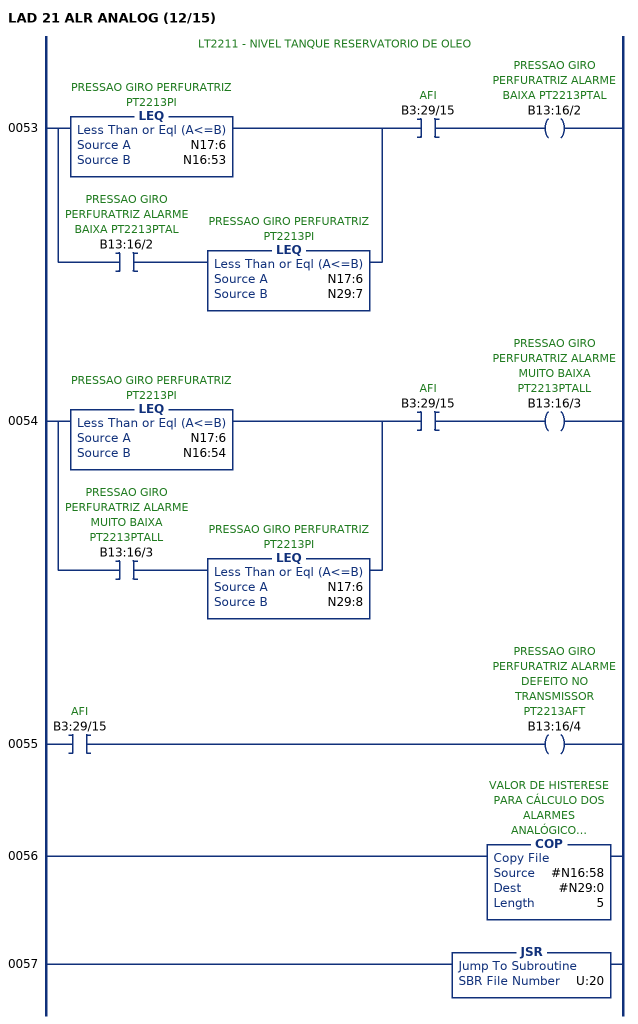
% Rung: 53 %
% LT2211 - NIVEL TANQUE RESERVATORIO DE OLEO %
SOR BST LEQ N17:6 N16:53 NXB XIC B13:16/2 LEQ N17:6 N29:7 BND XIC B3:29/15 OTE B13:16/2 EOR
%   N17:6  PT2213PI  "PRESSAO GIRO PERFURATRIZ" %
%   N16:53  PT2213L  "PRESSAO GIRO PERFURATRIZ BAIXA" %
%   B13:16/2  PT2213PTAL  "PRESSAO GIRO PERFURATRIZ ALARME BAIXA" %
%   N29:7  LIM_AL_L  "LIMITE PARA PERMITIR O REARME DO ALARME L (BAIXO)" %
%   B3:29/15  AFI %
% Rung: 54 %
SOR BST LEQ N17:6 N16:54 NXB XIC B13:16/3 LEQ N17:6 N29:8 BND XIC B3:29/15 OTE B13:16/3 EOR
%   N17:6  PT2213PI  "PRESSAO GIRO PERFURATRIZ" %
%   N16:54  PT2213LL  "PRESSAO GIRO PERFURATRIZ MUITO BAIXA" %
%   B13:16/3  PT2213PTALL  "PRESSAO GIRO PERFURATRIZ ALARME MUITO BAIXA" %
%   N29:8  LIM_AL_LL  "LIMITE PARA PERMITIR O REARME DO ALARME LL (MUITO BAIXO)" %
%   B3:29/15  AFI %
% Rung: 55 %
SOR XIC B3:29/15 OTE B13:16/4 EOR
%   B3:29/15  AFI %
%   B13:16/4  PT2213AFT  "PRESSAO GIRO PERFURATRIZ ALARME DEFEITO NO TRANSMISSOR" %
% Rung: 56 %
SOR COP #N16:58 #N29:0 5 EOR
%   N16:58  LT2211HIS  "NIVEL TANQUE OLEO HISTERESE" %
%   N29:0  HISTERESE  "VALOR DE HISTERESE PARA CÁLCULO DOS ALARMES ANALÓGICOS" %
% Rung: 57 %
SOR JSR U:20 EOR

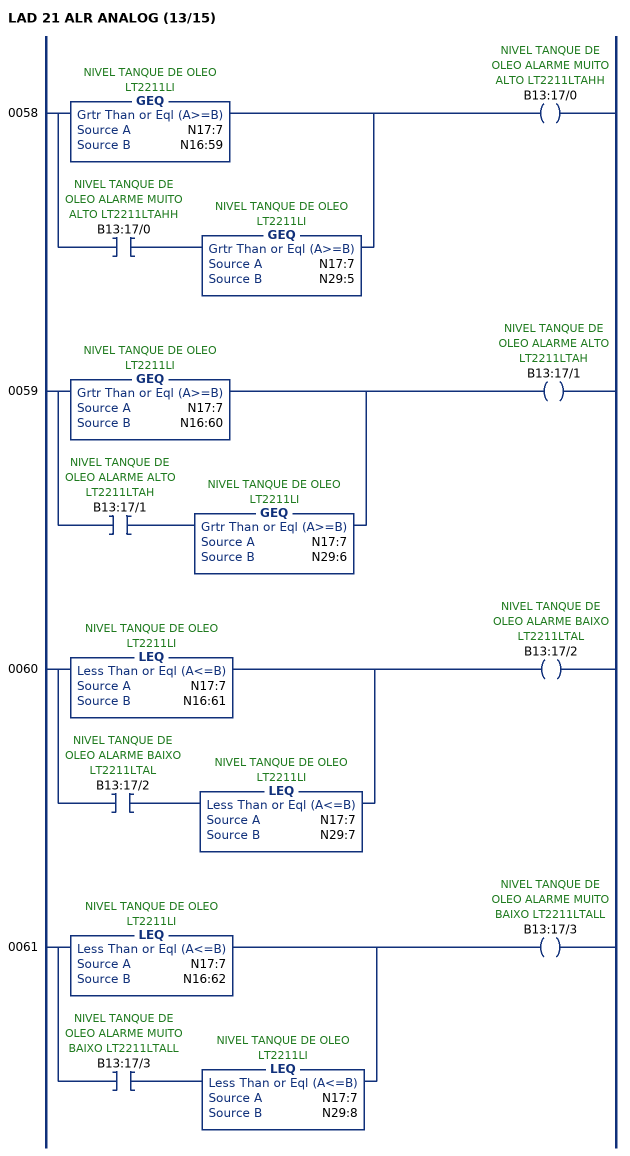
% Rung: 58 %
SOR BST GEQ N17:7 N16:59 NXB XIC B13:17/0 GEQ N17:7 N29:5 BND OTE B13:17/0 EOR
%   N17:7  LT2211LI  "NIVEL TANQUE DE OLEO" %
%   N16:59  LT2211HH  "NIVEL TANQUE OLEO MUITO ALTO" %
%   B13:17/0  LT2211LTAHH  "NIVEL TANQUE DE OLEO ALARME MUITO ALTO" %
%   N29:5  LIM_AL_HH  "LIMITE PARA PERMITIR O REARME DO ALARME HH (MUITO ALTO)" %
% Rung: 59 %
SOR BST GEQ N17:7 N16:60 NXB XIC B13:17/1 GEQ N17:7 N29:6 BND OTE B13:17/1 EOR
%   N17:7  LT2211LI  "NIVEL TANQUE DE OLEO" %
%   N16:60  LT2211H  "NIVEL TANQUE OLEO ALTO" %
%   B13:17/1  LT2211LTAH  "NIVEL TANQUE DE OLEO ALARME ALTO" %
%   N29:6  LIM_AL_H  "LIMITE PARA PERMITIR O REARME DO ALARME H (ALTO)" %
% Rung: 60 %
SOR BST LEQ N17:7 N16:61 NXB XIC B13:17/2 LEQ N17:7 N29:7 BND OTE B13:17/2 EOR
%   N17:7  LT2211LI  "NIVEL TANQUE DE OLEO" %
%   N16:61  LT2211L  "NIVEL TANQUE OLEO BAIXO" %
%   B13:17/2  LT2211LTAL  "NIVEL TANQUE DE OLEO ALARME BAIXO" %
%   N29:7  LIM_AL_L  "LIMITE PARA PERMITIR O REARME DO ALARME L (BAIXO)" %
% Rung: 61 %
SOR BST LEQ N17:7 N16:62 NXB XIC B13:17/3 LEQ N17:7 N29:8 BND OTE B13:17/3 EOR
%   N17:7  LT2211LI  "NIVEL TANQUE DE OLEO" %
%   N16:62  LT2211LL  "NIVEL TANQUE OLEO MUITO BAIXO" %
%   B13:17/3  LT2211LTALL  "NIVEL TANQUE DE OLEO ALARME MUITO BAIXO" %
%   N29:8  LIM_AL_LL  "LIMITE PARA PERMITIR O REARME DO ALARME LL (MUITO BAIXO)" %

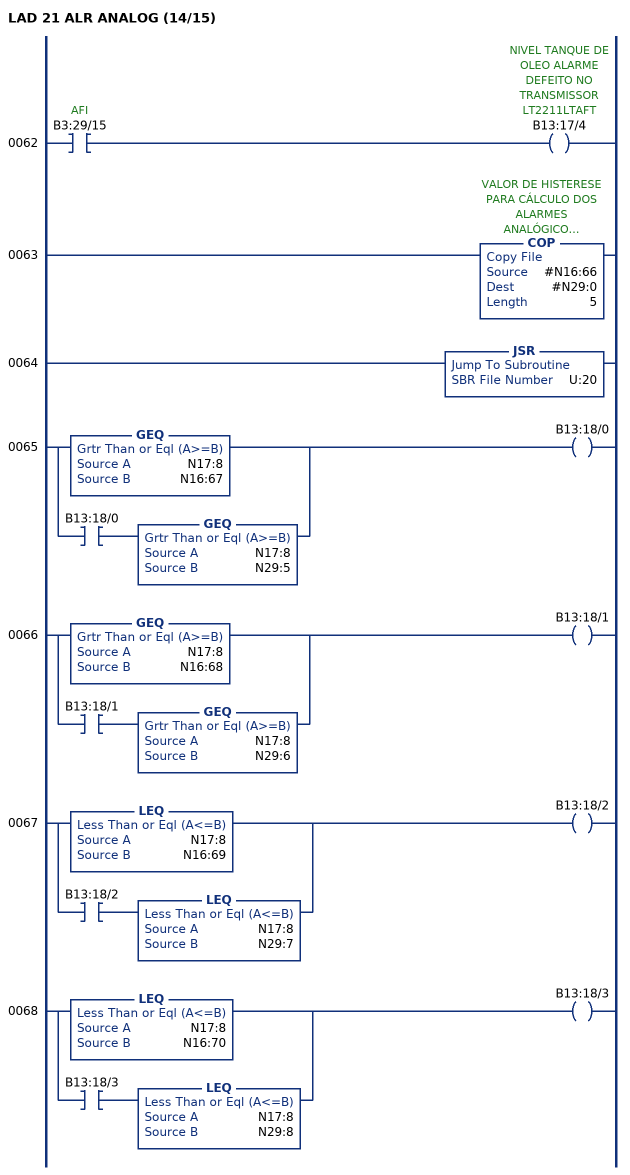
% Rung: 62 %
SOR XIC B3:29/15 OTE B13:17/4 EOR
%   B3:29/15  AFI %
%   B13:17/4  LT2211LTAFT  "NIVEL TANQUE DE OLEO ALARME DEFEITO NO TRANSMISSOR" %
% Rung: 63 %
SOR COP #N16:66 #N29:0 5 EOR
%   N29:0  HISTERESE  "VALOR DE HISTERESE PARA CÁLCULO DOS ALARMES ANALÓGICOS" %
% Rung: 64 %
SOR JSR U:20 EOR
% Rung: 65 %
SOR BST GEQ N17:8 N16:67 NXB XIC B13:18/0 GEQ N17:8 N29:5 BND OTE B13:18/0 EOR
%   N29:5  LIM_AL_HH  "LIMITE PARA PERMITIR O REARME DO ALARME HH (MUITO ALTO)" %
% Rung: 66 %
SOR BST GEQ N17:8 N16:68 NXB XIC B13:18/1 GEQ N17:8 N29:6 BND OTE B13:18/1 EOR
%   N29:6  LIM_AL_H  "LIMITE PARA PERMITIR O REARME DO ALARME H (ALTO)" %
% Rung: 67 %
SOR BST LEQ N17:8 N16:69 NXB XIC B13:18/2 LEQ N17:8 N29:7 BND OTE B13:18/2 EOR
%   N29:7  LIM_AL_L  "LIMITE PARA PERMITIR O REARME DO ALARME L (BAIXO)" %
% Rung: 68 %
SOR BST LEQ N17:8 N16:70 NXB XIC B13:18/3 LEQ N17:8 N29:8 BND OTE B13:18/3 EOR
%   N29:8  LIM_AL_LL  "LIMITE PARA PERMITIR O REARME DO ALARME LL (MUITO BAIXO)" %

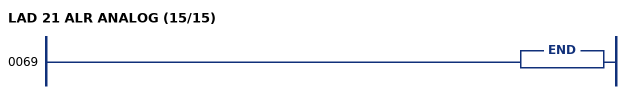
% Rung: 69 %
SOR END EOR

LADDER 22 "UNID ENG"
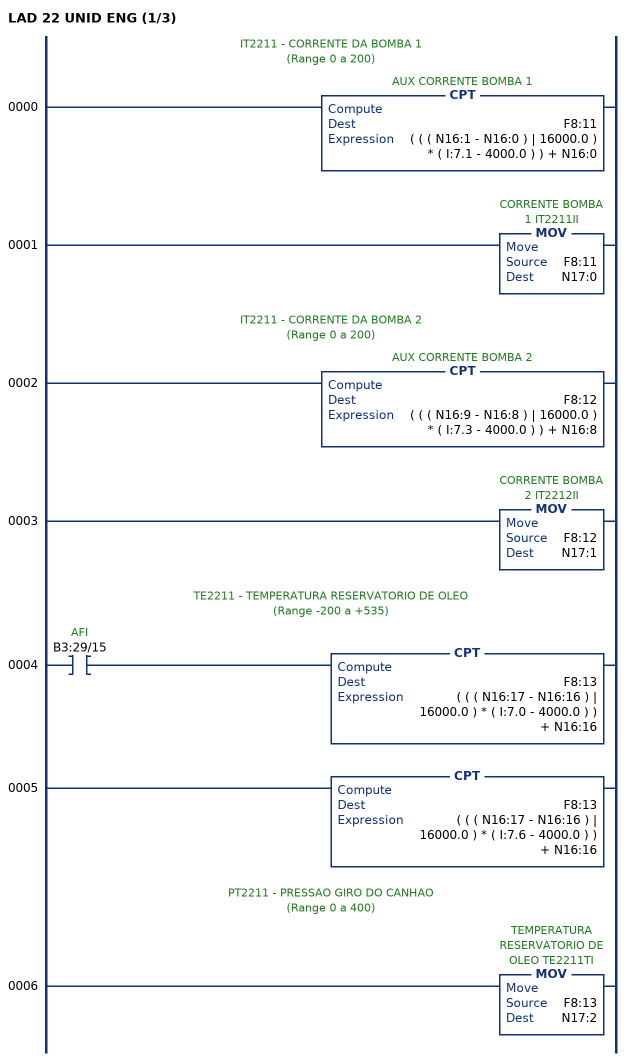
% Rung: 0 %
% IT2211 - CORRENTE DA BOMBA 1
% (Range 0 a 200) %
SOR CPT F8:11 " ( ( ( N16:1 - N16:0 ) | 16000.0 ) * ( I:7.1 - 4000.0 ) ) + N16:0 " EOR
%   F8:11  "AUX CORRENTE BOMBA 1" %
%   N16:1  IT2211MAX  "CORRENTE BOMBA 1 MAXIMO" %
%   N16:0  IT2211MIN  "CORRENTE BOMBA 1 MINIMO" %
%   I:7.1  MT2211  "MOTOR BOMBA 1 MEDICAO DE CORRENTE" %
% Rung: 1 %
SOR MOV F8:11 N17:0 EOR
%   F8:11  "AUX CORRENTE BOMBA 1" %
%   N17:0  IT2211II  "CORRENTE BOMBA 1" %
% Rung: 2 %
% IT2211 - CORRENTE DA BOMBA 2
% (Range 0 a 200) %
SOR CPT F8:12 " ( ( ( N16:9 - N16:8 ) | 16000.0 ) * ( I:7.3 - 4000.0 ) ) + N16:8 " EOR
%   F8:12  "AUX CORRENTE BOMBA 2" %
%   N16:9  IT2212MAX  "CORRENTE BOMBA 2 MAXIMO" %
%   N16:8  IT2212MIN  "CORRENTE BOMBA 2 MINIMO" %
%   I:7.3  MT2213  "MOTOR BOMBA 2 MEDICAO DE CORRENTE" %
% Rung: 3 %
SOR MOV F8:12 N17:1 EOR
%   F8:12  "AUX CORRENTE BOMBA 2" %
%   N17:1  IT2212II  "CORRENTE BOMBA 2" %
% Rung: 4 %
% TE2211 - TEMPERATURA RESERVATORIO DE OLEO
% (Range -200 a +535) %
SOR XIC B3:29/15 CPT F8:13 " ( ( ( N16:17 - N16:16 ) | 16000.0 ) * ( I:7.0 - 4000.0 ) ) + N16:16 " EOR
%   B3:29/15  AFI %
%   N16:17  TE2211MAX  "TEMPERATURA RESERVATORIO DE OLEO MAXIMO" %
%   N16:16  TE2211MIN  "TEMPERATURA RESERVATORIO DE OLEO MINIMO" %
%   I:7.0  TE2211  "TEMPERATURA RESERVATORIO DE OLEO" %
% Rung: 5 %
SOR CPT F8:13 " ( ( ( N16:17 - N16:16 ) | 16000.0 ) * ( I:7.6 - 4000.0 ) ) + N16:16 " EOR
%   N16:17  TE2211MAX  "TEMPERATURA RESERVATORIO DE OLEO MAXIMO" %
%   N16:16  TE2211MIN  "TEMPERATURA RESERVATORIO DE OLEO MINIMO" %
%   I:7.6  FT2211  "TRANSMISSOR DE VOLUME LAMA INJETADO" %
% Rung: 6 %
% PT2211 - PRESSAO GIRO DO CANHAO
% (Range 0 a 400) %
SOR MOV F8:13 N17:2 EOR
%   N17:2  TE2211TI  "TEMPERATURA RESERVATORIO DE OLEO" %

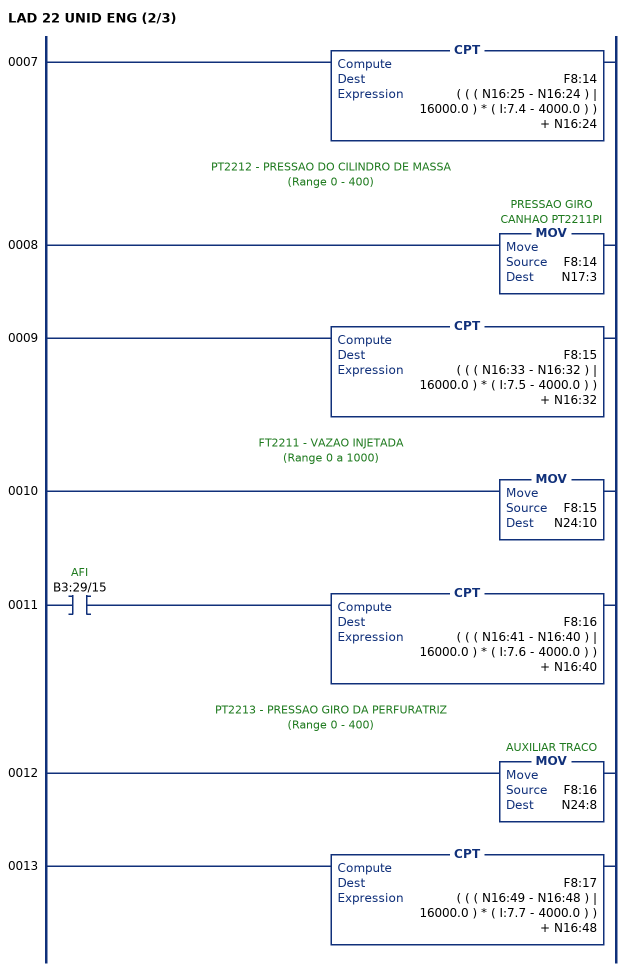
% Rung: 7 %
SOR CPT F8:14 " ( ( ( N16:25 - N16:24 ) | 16000.0 ) * ( I:7.4 - 4000.0 ) ) + N16:24 " EOR
%   N16:25  PT2211MAX  "GIRO CANHAO PRESSAO MAXIMO" %
%   N16:24  PT2211MIN  "GIRO CANHAO PRESSAO MINIMO" %
%   I:7.4  PT2211  "TRANSMISSOR DE PRESSAO DE GIRO DO CANHAO" %
% Rung: 8 %
% PT2212 - PRESSAO DO CILINDRO DE MASSA
% (Range 0 - 400) %
SOR MOV F8:14 N17:3 EOR
%   N17:3  PT2211PI  "PRESSAO GIRO CANHAO" %
% Rung: 9 %
SOR CPT F8:15 " ( ( ( N16:33 - N16:32 ) | 16000.0 ) * ( I:7.5 - 4000.0 ) ) + N16:32 " EOR
%   N16:33  PT2212MAX  "CILINDRO MASSA CANHAO PRESSAO MAXIMO" %
%   N16:32  PT2212MIN  "CILINDRO MASSA CANHAO PRESSAO MINIMO" %
%   I:7.5  PT2212  "TRANSMISSOR DE PRESSAO CILINDRO DE MASSA CANHAO" %
% Rung: 10 %
% FT2211 - VAZAO INJETADA
% (Range 0 a 1000) %
SOR MOV F8:15 N24:10 EOR
% Rung: 11 %
SOR XIC B3:29/15 CPT F8:16 " ( ( ( N16:41 - N16:40 ) | 16000.0 ) * ( I:7.6 - 4000.0 ) ) + N16:40 " EOR
%   B3:29/15  AFI %
%   N16:41  FT2211MAX  "TRACO INJETADO VAZAO MAXIMO" %
%   N16:40  FT2211MIN  "TRACO INJETADO VAZAO MINIMO" %
%   I:7.6  FT2211  "TRANSMISSOR DE VOLUME LAMA INJETADO" %
% Rung: 12 %
% PT2213 - PRESSAO GIRO DA PERFURATRIZ
% (Range 0 - 400) %
SOR MOV F8:16 N24:8 EOR
%   N24:8  "AUXILIAR TRACO" %
% Rung: 13 %
SOR CPT F8:17 " ( ( ( N16:49 - N16:48 ) | 16000.0 ) * ( I:7.7 - 4000.0 ) ) + N16:48 " EOR
%   N16:49  PT2213MAX  "PRESSAO GIRO PERFURATRIZ MAXIMO" %
%   N16:48  PT2213MIN  "PRESSAO GIRO PERFURATRIZ MINIMO" %
%   I:7.7  PT2213  "TRANSMISSOR DE PRESSAO GIRO PERFURATRIZ" %

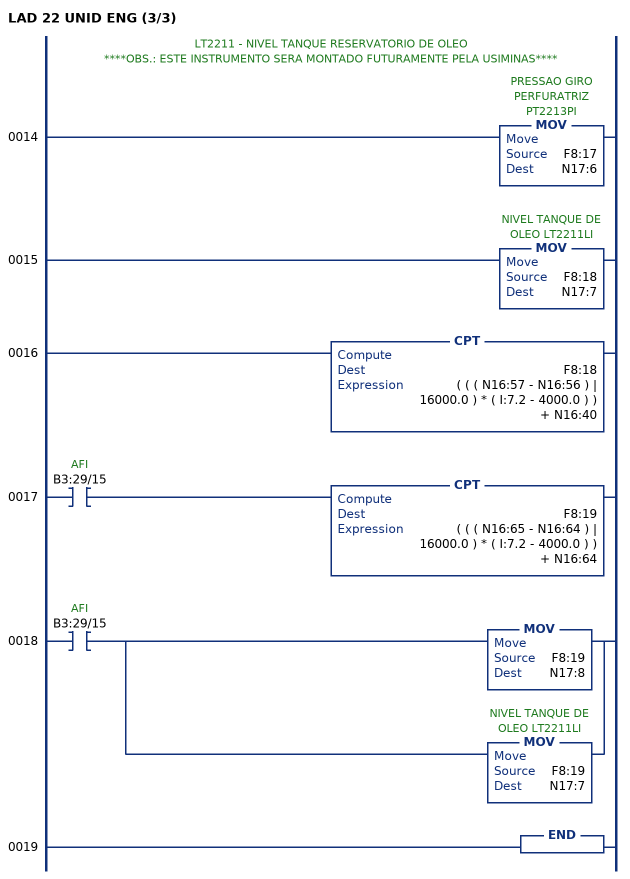
% Rung: 14 %
% LT2211 - NIVEL TANQUE RESERVATORIO DE OLEO
% ****OBS.: ESTE INSTRUMENTO SERA MONTADO FUTURAMENTE PELA USIMINAS**** %
SOR MOV F8:17 N17:6 EOR
%   N17:6  PT2213PI  "PRESSAO GIRO PERFURATRIZ" %
% Rung: 15 %
SOR MOV F8:18 N17:7 EOR
%   N17:7  LT2211LI  "NIVEL TANQUE DE OLEO" %
% Rung: 16 %
SOR CPT F8:18 " ( ( ( N16:57 - N16:56 ) | 16000.0 ) * ( I:7.2 - 4000.0 ) ) + N16:40 " EOR
%   N16:57  LT2211MAX  "NIVEL TANQUE OLEO MAXIMO" %
%   N16:56  LT2211MIN  "NIVEL TANQUE OLEO MINIMO" %
%   N16:40  FT2211MIN  "TRACO INJETADO VAZAO MINIMO" %
% Rung: 17 %
SOR XIC B3:29/15 CPT F8:19 " ( ( ( N16:65 - N16:64 ) | 16000.0 ) * ( I:7.2 - 4000.0 ) ) + N16:64 " EOR
%   B3:29/15  AFI %
% Rung: 18 %
SOR XIC B3:29/15 BST MOV F8:19 N17:8 NXB MOV F8:19 N17:7 BND EOR
%   B3:29/15  AFI %
%   N17:7  LT2211LI  "NIVEL TANQUE DE OLEO" %
% Rung: 19 %
SOR END EOR

LADDER 23 "RESET"    % Reset geral para 1 scan %
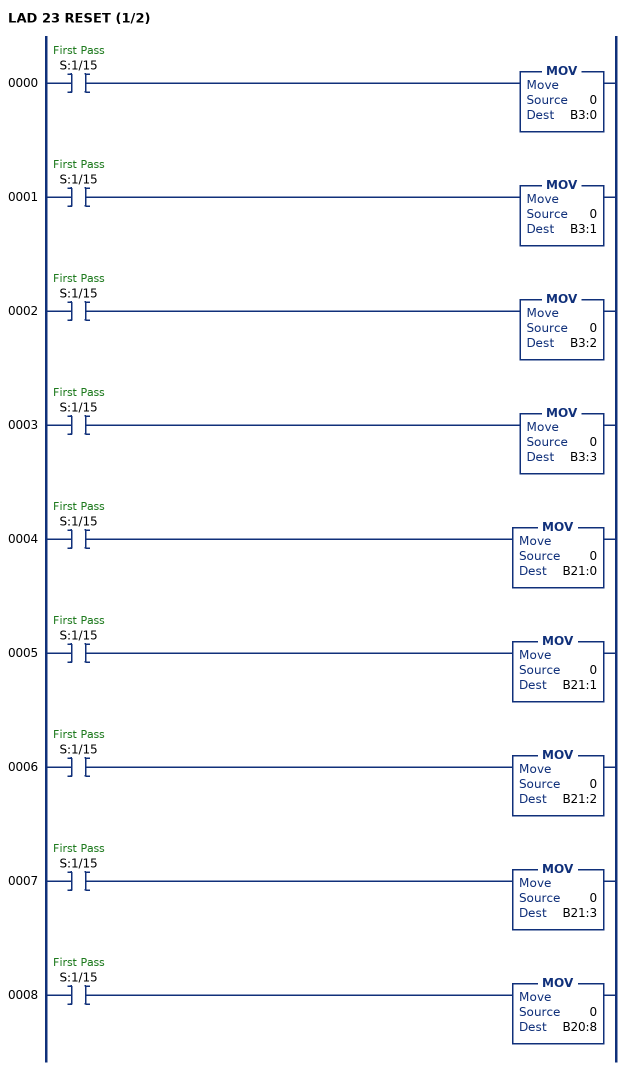
% Rung: 0 %
SOR XIC S:1/15 MOV 0 B3:0 EOR
%   S:1/15  "First Pass" %
% Rung: 1 %
SOR XIC S:1/15 MOV 0 B3:1 EOR
%   S:1/15  "First Pass" %
% Rung: 2 %
SOR XIC S:1/15 MOV 0 B3:2 EOR
%   S:1/15  "First Pass" %
% Rung: 3 %
SOR XIC S:1/15 MOV 0 B3:3 EOR
%   S:1/15  "First Pass" %
% Rung: 4 %
SOR XIC S:1/15 MOV 0 B21:0 EOR
%   S:1/15  "First Pass" %
% Rung: 5 %
SOR XIC S:1/15 MOV 0 B21:1 EOR
%   S:1/15  "First Pass" %
% Rung: 6 %
SOR XIC S:1/15 MOV 0 B21:2 EOR
%   S:1/15  "First Pass" %
% Rung: 7 %
SOR XIC S:1/15 MOV 0 B21:3 EOR
%   S:1/15  "First Pass" %
% Rung: 8 %
SOR XIC S:1/15 MOV 0 B20:8 EOR
%   S:1/15  "First Pass" %

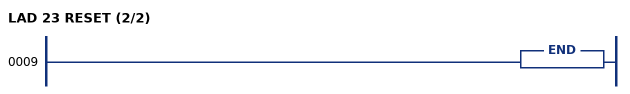
% Rung: 9 %
SOR END EOR

OTHER DOCUMENTED ADDRESSES
  B3:0/7  "AUXILIAR"
  B3:0/8  "AUXILIAR PUSO LOCAL-MESA"
  B3:0/9  "AUXILIAR"
  B3:0/10  "AUXILIAR PUSO MESA-LOCAL"
  B3:1/7  "AUXILIAR"
  B3:1/8  "AUX PULSO LOCAL-MESA"
  B3:1/9  "AUXILIAR"
  B3:1/10  "AUX PULSO MESA-LOCAL"
  B3:2/7  "AUXILIAR"
  B3:2/8  "AUXILIAR PUSO LOCAL-MESA"
  B3:2/9  "AUXILIAR"
  B3:2/10  "AUXILIAR PUSO MESA-LOCCAL"
  B3:3/7  "AUXILIAR DESATIVA BOMBA"
  B3:21/3  "AUXILIAR CHEGADA POSICAO REPOUSO"
  B3:26/1  "AUX CHAVE RESERV OLEO NIVEL BAIXO"
  B3:29/3  H_B11_E02  "HABILITA O ENVIO DA MSG DO ARQUIVO DE ESTADOS (B11) PARA A ESTAÇÃO DE OPERAÇÃO Nº2 (EO2)"
  B3:29/4  H_B11_E03  "HABILITA O ENVIO DA MSG DO ARQUIVO DE ESTADOS (B11) PARA A ESTAÇÃO DE OPERAÇÃO Nº3 (EO3)"
  B3:29/5  H_B11_ALPHA  "HABILITA O ENVIO DA MSG DO ARQUIVO DE ESTADOS (B11) PARA O ALPHA DIGITAL"
  B10:0/0  E_MT2211TLI  "BOMBA 1 COMANDO LIGA"
  B10:0/1  E_MT2211TDL  "BOMBA 1 COMANDO DESLIGA"
  B10:0/3  E_1B4MC2211TLI  "MESA BOTAO LIGA BOMBA"
  B10:0/4  E_1B5MC2211TDL  "MESA BOTAO DESLIGA BOMBA"
  B10:0/6  E_MT2213TLI  "BOMBA 2 COMANDO LIGA"
  B10:0/7  E_MT2213TDL  "BOMBA 2 COMANDO DESLIGA"
  B10:0/9  E_1B6MC2211TLI  "MESA BOMBA 2 BOTAO LIGA"
  B10:0/10  E_1B7MC2211TDL  "MESA BOMBA 2 BOTAO DESLIGA"
  B10:0/12  E_MT2212TLI  "BOMBA REFRIGERACAO 1 COMANDO LIGA"
  B10:0/13  E_MT2212TDL  "BOMBA REFRIGERACAO 1 COMANDO DESLIGA"
  B10:1/2  E_MT2231TLI  "BOMBA AGUA REFRIG BROCA 1 COMANDO LIGA"
  B10:1/3  E_MT2231TDL  "BOMBA AGUA REFRIG BROCA 1 COMANDO DESLIGA"
  B10:3/6  E_BZ2221TLI  "SIRENE COMANDO LIGA"
  B10:4/0  E_MT2211SLIC  "BOMBA 1 CONTATOR FECHADO"
  B10:4/2  E_MT2211SDLC  "BOMBA 1 DISJUNTOR LIGADO"
  B10:4/10  E_MT2213SLIC  "BOMBA 2 CONTATOR FECHADO"
  B10:4/12  E_MT2213SDLC  "BOMBA 2 DISJUNTOR LIGADO"
  B10:5/5  E_MT2212SLIC  "BOMBA REFRIGERACAO 1 LIGADO"
  B10:5/7  E_MT2212SDLC  "BOMBA REFRIGERACAO 1 DISJUNTOR LIGADO"
  B10:6/0  E_MT2231SLIC  "BOMBA AGUA REFRIG BROCA 1 CONTATOR FECHADO"
  B10:6/2  E_MT2231SDLC  "BOMBA AGUA REFRIG BROCA 1 DISJUNTOR LIGADO"
  B10:6/10  E_ZS2211LPF  "VALVULA SUCCAO BOMBA REFRIG POS FECHADA"
  B10:6/12  E_ZS2212LPF  "VALV SUCCAO BOMBA 1 POSICAO FECHADA"
  B10:6/14  E_ZS2213LPF  "VALV SUCCAO BOMBA 2 POSICAO FECHADA"
  B10:7/0  E_MT2211SSCC  "BOMBA 1 SOBRECARGA"
  B10:7/1  E_MT2211AFCF  "BOMBA PRINCIPAL 1 FALHA NO CONTATOR FECHAMENTO"
  B10:7/2  E_MT2211SDAT  "BOMBA 1 DISJUNTOR EM TRIP"
  B10:7/4  E_MT2213SSCC  "BOMBA 2 SOBRECARGA"
  B10:7/5  E_MT2213AFCF  "BOMBA RESERVA 1 FALHA NO CONTATOR FECHAMENTO"
  B10:7/6  E_MT2213SDAT  "BOMBA 2 DISJUNTOR EM TRIP"
  B10:7/8  E_MT2212SSCC  "BOMBA REFRIGERACAO 1 SOBRECARGA"
  B10:7/9  E_MT2212AFCF  "BOMBA REFRIGERACAO 1 FALHA NO CONTATOR FECHAMENTO"
  B10:7/10  E_MT2212SDAT  "BOMBA REFRIGERACAO 1 DISJUNTOR EM TRIP"
  B10:7/12  E_MT2231SSCC  "BOMBA AGUA REFRIG BROCA 1 SOBRECARGA"
  B10:7/13  E_MT2231AFCF  "BOMBA AGUA REFRIG BROCA 1 FALHA CONTATOR FECHAMENTO"
  B10:7/14  E_MT2231SDAT  "BOMBA AGUA REFRIG BROCA 1 DISJUNTOR EM TRIP"
  B10:8/0  E_LSH2211LAH  "CHAVE RESERV OLEO NIVEL ALTO"
  B10:8/2  E_LSL2212LAL  "CHAVE RESERV OLEO NIVEL BAIXO"
  B10:8/4  E_LSLL2213LTAL  "CHAVE RESERV OLEO NIVEL MUITO BAIXO"
  B10:8/6  E_PDS2211PAL  "PRESSOSTATO DIF FILTRO RESERV 1 PRESSÃO BAIXA"
  B10:8/8  E_PDS2212PAL  "PRESSOSTATO DIF FILTRO RESERV 2 PRESSÃO BAIXA"
  B10:8/10  E_PDS2213PAL  "PRESSOSTATO DIF FILTRO RESERV 3 PRESSÃO BAIXA"
  B10:8/12  E_PDS2214PAL  "PRESSOSTATO DIF FILTRO RESERV 4 PRESSÃO BAIXA"
  B10:8/14  E_PDS2215PAL  "PRESSOSTATO DIF FILTRO RESERV 5 PRESSÃO BAIXA"
  B10:9/0  E_PDS2216PAL  "PRESSOSTATO DIF FILTRO RESERV 6 PRESSÃO BAIXA"
  B10:9/2  E_PS2211PAL  "PRESSOSTATO BOMBA 1 PRESSAO BAIXA"
  B10:9/4  E_PS2212PAL  "PRESSOSTATO BOMBA 2 PRESSAO BAIXA"
  B10:9/6  E_PSH2214PAL  "PRESSOSTATO CANHAO FURO COR. PRESSÃO ALTA"
  B10:9/8  E_PS2231PAL  "PRESSOSTATO LINHA AR COMPRIMIDO PRESSÃO BAIXA"
  B10:9/10  E_FS2231FAL  "CHAVE FLUXO LINHA AR RESF BROCA PRESSÃO BAIXA"
  B10:11/0  E_1U1SLIC  "FONTE 24VCC FUNCIONANDO"
  B10:11/2  E_1A1SLIC  "DISJUNTOR GERAL LIGADO"
  B10:11/4  E_1E8AFF  "RELE FALTA DE FASE ATUADO"
  B10:11/6  E_1B1CL2212SLFRC  "CILINDRO DE MASSA AVANCO LOCAL"
  B10:11/8  E_1B2CL2212SLRC  "CILINDRO DE MASSA RECUO LOCAL"
  B10:11/10  E_1S1CL2212LLOC  "SELECAO MOV DO CILINDRO DE MASSA MODO LOCAL"
  B10:11/12  E_1S1CL2212LREM  "SELECAO MOV DO CILINDRO DE MASSA MODO MESA"
  B10:12/0  E_1S1MC2211LLI  "MANETE CONTROLE DO GIRO CANHAO PARA BOCA"
  B10:12/2  E_1S1MC2211LPS  "MANETE CONTROLE DO GIRO DO CANHAO POSICAO REPOUSO"
  B10:12/4  E_1S2MC2211SLFRC  "MANETE CONTROLE DE INJECAO DE MASSA POSICAO AVANÇO"
  B10:12/6  E_1S2MC2211SLRC  "MANETE CONTROLE DE INJECAO DE MASSA POSICAO RECUO"
  B10:12/8  E_1S3MC2211LLOC  "CHAVE SELETORA CANHAO POSICAO LOCAL"
  B10:12/12  E_1B1MC2211BLIP  "CANHAO BOTAO HABILITA INJECAO DE MASSA"
  B10:12/14  E_1B2MC2211BLIP  "CANHAO ALERTA DE MOVIMENTO BOTAO LIGA SIRENE"
  B10:13/0  E_1B3MC2211BLIP  "TESTE LAMPADA BOTAO LIGA"
  B10:13/2  E_1B3MC2211LLL1  "UNIDADE HID CHAVE SELETORA LOCAL"
  B10:13/6  E_1S5MC2211LLL1  "UNIDADE HID SELECAO BOMBA 1"
  B10:13/10  E_1B8MC2211BLIP  "BOTAO REARME CANHAO E UNID HIDRAULICA"
  B10:13/12  E_1S6MC2211LLI  "MANETE CONTROLE DESLOCAMENTO PERFURATRIZ PARA BOCA"
  B10:13/14  E_1S6MC2211LPS  "MANETE CONTROLE DESLOCAMENTO PERFURATRIZ REPOUSO"
  B10:14/0  E_1S7MC2211SLBVC  "MANETE CARRO AVANCO 1"
  B10:14/2  E_1S7MC2211SLAVC  "MANETE CARRO AVANCO 2"
  B10:14/4  E_1S7MC2211SLRC  "MANETE CARRO RECUO"
  B10:14/6  E_1S8MC2211SLFRC  "MANETE MARRETA DE IMPACTO A FRENTE"
  B10:14/8  E_1S8MC2211SLRC  "MANETE MARRETA DE IMPACTO REVERSO"
  B10:14/10  E_1S9MC2211SLIC  "SELETORA LIGA GIRO DA BROCA"
  B10:14/12  E_1S10MC2211SLIC  "SELETORA LIGA SOPRO REFRIGERACAO"
  B10:14/14  E_1S11MC2211SPL1L  "SELETORA DA BROCA MISTURA"
  B10:15/2  E_1B9MC2211TLI  "PERFURATRIZ BOTAO ATIVA SIRENE"
  B10:15/4  E_1B10MC2211TRE  "BOTAO REARME PERFURATRIZ"
  B10:15/6  E_1B11MC2211TRE  "PERFURATRIZ/CANHAO BOTAO RECONHECE ALARME"
  B20:0/0  E_MT2211CLIC  "BOMBA 1 LIGAR"
  B20:1/0  E_MT2213CLIC  "BOMBA 2 LIGAR"
  B20:2/0  E_MT2212CLIC  "BOMBA REFRIGERACAO LIGAR"
  B20:3/0  E_MT2231CLIC  "BOMBA AGUA REFRIG BROCA 1 LIGAR"
  B20:4/4  E_VS2211ACLAC  "VALV PROP GIRO CANHAO AVANCO LIGA ABRIR"
  B20:4/5  E_VS2211BCLAC  "VALV PROP GIRO CANHAO RETORNO LIGA ABRIR"
  B20:4/8  E_VS2212ACLAC  "VALV PROP CILINDRO CANHAO LIGA ABRIR AVANCO"
  B20:4/9  E_VS2212BCLAC  "VALV PROP CILINDRO CANHAO LIGA ABRIR RETORNO"
  B20:4/12  E_VS2214CLAC  "VALV DIRECIONAL BLOQ GIRO CANHAO LIGA ABRIR"
  B20:5/0  E_VS2213ACLAC  "VALV PROP GIRO PERF LIGA ABRIR AVANCO"
  B20:5/1  E_VS2213BCLAC  "VALV PROP GIRO PERF LIGA ABRIR RETORNO"
  B20:5/4  E_VS2216CLAC  "VALV DIREC BLOQ GIRO PERF LIGA ABRIR"
  B20:5/8  E_VS2217ACLAC  "VALV TRAVA GIRO PERFURATRIZ LIGA ABRIR"
  B20:5/10  E_VS2217BCLAC  "VALV DISTRAVA GIRO PERFURATRIZ LIGA ABRIR"
  B20:5/12  E_VS2231CLAC  "VALV DIREC RECUO MOTOR TRANS LIGA ABRIR"
  B20:6/0  E_VS2232CLAC  "VALV DIREC AVANCO MOTOR TRANS LIGA ABRIR"
  B20:6/4  E_VS2233CLAC  "VALV DIREC BLOQ AVAN MOTOR TRANS LIGA ABRIR"
  B20:6/8  E_VS2234CLAC  "VALV DIRECIONAL MARTELO A FRENTE LIGA ABRIR"
  B20:6/12  E_VS2235CLAC  "VALV DIRECIONAL MARTELO A TRAS LIGA ABRIR"
  B20:7/0  E_VS2236CLAC  "VALV DIRECIONAL GIRO DA BROCA LIGA ABRIR"
  B20:7/4  E_VS2237CLAC  "VALV DIREC RESF BROCA LIGA ABRIR"
  B20:7/8  E_VS2238CLAC  "VALV DIREC AGUA RESF BROCA LIGA ABRIR"
  B20:7/12  E_BZ2211CLIC  "SIRENE LIGAR"
  B20:8/0  "ALARME SONORO MESA"
  B20:8/1  E_LCPRCLAC  "LAMPADA CANHAO POSICAO REPOUSO LIGAR"
  B20:8/2  E_1H1CLAC  "LAMPADA PRESSAO DO CANHAO NA BOCA OK"
  B20:8/4  E_1H2CLAC  "LAMPADA INJECAO DE MASSA NO CAMPO"
  B20:8/6  E_1H3CLAC  "LAMPADA CANHAO NA POSICAO REPOUSO"
  B20:8/8  E_1H4CLAC  "LAMPADA BOMBA 1 LIGADA"
  B20:8/10  E_1H5CLAC  "LAMPADA BOMBA 2 LIGADA"
  B20:8/12  E_1H6CLAC  "LAMPADA PRESSAO HIDRAULICA OK"
  B20:8/14  E_1H7CLAC  "MATRIZ 1 LAMPADA NIVEL TANQUE OLEO ALTO"
  B20:9/0  E_1H8CLAC  "MATRIZ 2 LAMPADA NIVEL TANQUE OLEO BAIXO"
  B20:9/2  E_1H9CLAC  "MATRIZ 3 LAMPADA NIVEL OLEO MUITO BAIXO"
  B20:9/4  E_1H10CLAC  "MATRIZ 4 LAMPADA BOMBA 1 DEFEITO"
  B20:9/6  E_1H11CLAC  "MATRIZ 5 LAMPADA BOMBA 2 DEFEITO"
  B20:9/8  E_1H12CLAC  "MATRIZ 6 LAMPADA BOMBA RECIRCULACAO DE OLEO DEFEITO"
  B20:9/10  E_1H13CLAC  "MATRIZ 7 LAMPADA TEMPERATURA OLEO ALTA"
  B20:9/12  E_1H14CLAC  "MATRIZ 8 LAMPADA FILTRO DE OLEO OBSTRUIDO"
  B20:9/14  E_1H15CLAC  "MATRIZ 9 LAMPADA PRESSAO INJECAO ALTA"
  B20:10/0  E_1H16CLAC  "MATRIZ 10 LAMPADA PRESSAO HIDRAULICA BOMBA 1/2 COM DEFEITO"
  B20:10/2  E_1H17CLAC  "MATRIZ 11 LAMPADA VALVULA ANTES BOMBA REFRIG FECHADA"
  B20:10/4  E_1H18CLAC  "MATRIZ 12 LAMPADA VALVULA MANUAL ANTES DA BOMBA 1 FECHADA"
  B20:10/6  E_1H19CLAC  "MATRIZ 13 LAMPADA VALVULA MANUAL ANTES DA BOMBA 2 FECHADA"
  B20:10/8  E_1H20CLAC  "MATRIZ 14 LAMPADA CHAVE DO PAINEL LOCAL ABASTEC EM LOCAL"
  B20:10/10  E_1H21CLAC  "MATRIZ 15"
  B20:10/12  E_1H22CLAC  "LAMPADA PRESSAO AR COMPRIMIDO BAIXA"
  B20:10/14  E_1H23CLAC  "LAMPADA REFRIGERACAO DA BROCA LIGADA"
  B20:11/0  E_1H24CLAC  "LAMPADA GIRO DA BROCA LIGADA"
  B20:11/2  E_1H25CLAC  "LAMPADA PERFURATRIZ TRAVADA CONTRA O FORNO"
  B20:11/4  E_1H26CLAC  "LAMPADA PERFURATRIZ POSICAO REPOUSO"
  B20:11/6  E_1H27CLAC  "MATRIZ 1 LAMPADA BOMBA DE AGUA REFRIG BROCA DEFEITO"
  B20:11/8  E_1H28CLAC  "MATRIZ 2 LAMPADA FLUXO AR/N2 REFRIG BROCA BAIXO"
  B20:11/10  E_1H29CLAC  "MATRIZ 3"
  B21:0/0  "AUXILIAR REARME DEFEITOS"
  B21:0/2  "Temporario"
  B33:0/10  "provisorio retirar apos teste"
  B33:0/11  "provisorio retirar apos teste"
  DFILE:0  "OUTPUT"
  DFILE:1  "INPUT"
  DFILE:2  "STATUS"
  DFILE:3  "BINARY"
  DFILE:4  "TIMER"
  DFILE:5  "COUNTER"
  DFILE:6  "CONTROL"
  DFILE:7  "INTEGER"
  DFILE:8  "FLOAT"
  DFILE:9  "COMANDO D"
  DFILE:10  "ESPELHO D Area Espelho entrada s e saidas digitais"
  DFILE:11  "STATUS Status do sistema qu e são enviados ao SS C"
  DFILE:13  "DEFEITO"
  DFILE:15  "ESPELHO A Area Espelho entrada s e saidas analogica s"
  DFILE:16  "SET POINT"
  DFILE:17  "LEITURA"
  DFILE:18  "COMANDO A"
  DFILE:21  "AUXILIARES auxiliares"
  I:3.0  "TE/TT-431601 TEMPERATURA DO GÁS DE ENTRADA DO VENTILADOR PRINCIPAL"
  I:3.0/0  "PSH2214 PRESSOSTATO CANHAO NO FURO PRESSAO ALTA"
  I:7.0/12  "VP VENTILADOR PRINCIPAL LIGADO"
  I:9.1/11  "MESA BOMBA 2 BOTAO LIGA"
  I:9.1/12  "MESA BOMBA 2 BOTAO DESLIGA"
  I:9.2/11  "PERFURATRIZ BOTAO ATIVA SIRENE"
  I:11.0/15  "CHAVE SELETORA CANHAO POSICAO MESA OPERACAO"
  I:12.0/6  "CHAVE SELETORA OPERAÇAO MESA"
  I:12.0/8  "SELECAO BOMBA 2"
  M00000:001.200  M0
  M10001:001.100  M1
  N26:60  B11_EO2  "ENVIO DOS ESTADOS PARA A ESTAÇÃO DE OPERAÇÃO Nº2"
  O:8.0  "VALV PROPORCIONAL GIRO DO CANAHO AVANCO RETORNO"
  O:9.6/1  "MATRIZ 15 2"
  O:9.6/10  "MATRIZ 3 2"
  PFILE:7  "Bomba Principal 1"
  PFILE:8  "Bomba Reserva 1"
  PFILE:19  "Comuinicao"
  T4:0  "TIMER GIRO C PARA CHEGADA NA POSICAO REPOUSO"
  T4:4  "TIMER GIRO C VALV PROPORCIONAL POSICAO AVANCO"
  T4:18  "TIMER PRESSAO ALTA"
  T4:19  "TIMER PRESSAO BAIXA"
  T4:20  "TIMER VAZAO ALTA"
  T4:21  "TIMER VAZAO BAIXA"
  T4:35  "TIMER DESLIGA BOMBA"
  T4:195  "TEMPO PARA ALARMAR PRESSÃO MUITO ALTA NA LINHA DE AR (ENTUPIMENTO)"
  T4:195/DN  "TEMPO PARA ALARMAR PRESSÃO MUITO ALTA NA LINHA DE AR (ENTUPIMENTO)"
  T4:198  "TEMPO PARA GARANTIR ALARME DE VIBRACAO PERMANECA POR MAIS DE 10 SEGUNDOS"
  T4:198/DN  "TEMPO PARA GARANTIR ALARME DE VIBRACAO PERMANECA POR MAIS DE 10 SEGUNDOS"
  T4:200  "TEMPO PARA ALARMAR PRESSÃO MUITO BAIXA NA LINHA DE AR (LINHA FURADA)"
  T20:42  TALVPIT  "TEMPO PARA HABILITAR ALARMES DE CORRENTE DO MOTOR DO VENTILADOR PRINCIPAL"
  U:26  "ARQUIVO DE CÁLCULO DA HISTERESE DOS ALARMES ANALÓGICOS"

COMMENTS NOT ATTACHED TO A CURRENT RUNG
  B13:3/2: SOBRECARGA
  B11:1/0: STATUS E DEFEITOS DOS EQUIPAMENTOS VINDOS DA AREA ESPELHO / =========================================================================================================
    BOMBA RESERVA - MT2213
    =========================================================================================================
  B11:0/5: CONDICOES DE PARTIDA DO EQUIPAMENTO
  O:0.0/0: COMANDO DOS EQUIPAMENTOS
  B10:0/0: AREA ESPELHO PARA ENTRADAS DIGITAIS
  B11:0/0: STATUS E DEFEITOS DOS EQUIPAMENTOS VINDOS DA AREA ESPELHO / =========================================================================================================
    BOMBA PRINCIPAL - MT2211
    =========================================================================================================
  N25:1: MOVE VALOR DE TRACO INJETADO PARA O DISPLAY
  B20:4/4: DESENERGIZACAO DA VALVULA NO INICIO DO MOVIMENTO DE RETORNO
  B20:7/12: SISTEMA DE CONTROLE DE GIRO DO CANHAO / MANETE POSICAO AVANCO ACIONA SIRENE POR 5s
    MANETE POSICAO RETORNO ACIONA SIRENE POR 2s
  N16:57: CONTROLE DA VELOCIDADE DE GIRO DO CANHAO
  B20:8/0: ESTAGIO FINAL
  T4:1: RETORNO DO CANHAO / COMANDO PARA RETORNO DO MOVIMENTO DA PERFURATRIZ
    RETORNO - APOS 2s ACIONA VALVULA PROPORCIONAL
  B3:0/11: *******************************************************************************************************
    CÁLCULO  DOS  LIMITES  DE  ALARME  ANALÓGICO  CONSIDERANDO  A  HISTERESE
    
    *******************************************************************************************************
  N17:50: MOVE O VALOR PARA O PONTO DE LEITURA
  B21:1/0: LAMPADA NIVEL OLEO  BAIXO
  B20:9/2: LAMPADA NIVEL OLEO MUITO BAIXO
  N16:56: ESTABILIDADE DA VELOCIDADE FINAL DO CANHAO
  T4:4: RAMPA DE SUBIDA
  B20:9/6: LAMPADA BOMBA 2 DEFEITO
  B20:9/8: LAMPADA BOMBA RECIRCULACAO DE OLEO DEFEITO
  B20:9/10: LAMPADA TEMPERATURA OLEO ALTA
  B21:1/10: LAMPADA TEMPERATURA OLEO ALTA
  B20:9/12: LAMPADA FILTRO DE OLEO OBSTRUIDO
  B20:9/14: LAMPADA PRESSAO INJECAO ALTA
  B20:10/2: LAMPADA VALVULA INTERLIGACAO RESERV ABERTA
  B20:11/8: LAMPADA FLUXO AR/N2 REFRIG BROCA BAIXA
  B3:62/8: **************************************************************************************************************************
    GERAÇÃO DE ALARMES DE VARIÁVEIS ANALÓGICAS CONSIDERANDO A HISTERESE
    *************************************************************************************************************************
  B13:9/0: CONTROLE DO MARTELETE DE PERFURACAO / PRESSOSTATO PS-2231
  B31:0/10: PULSO PARA DESLIGAR BOMBA QUANDO OCORRER MUDANCA NA SELECAO DA CHAVE
  B31:1/10: PULSO PARA DESLIGAR BOMBA QUANDO OCORRER MUDANCA NA SELECAO DA CHAVE
  B31:2/10: PULSO PARA DESLIGAR BOMBA QUANDO OCORRER MUDANCA NA SELECAO DA CHAVE
  B31:19/1: POSICAO REPOUSO DA PERFURATRIZ
  B31:22/1: CANHAO POSICAO REPOUSO
  B20:10/4: LIGA ROTATOR
  B20:4/9: RECUO
  O:8.0: MOVE VALOR PARA SAIDA ANALOGICA DA VALVULA VS2211
  O:8.1: MOVE VALOR PARA SAIDA ANALOGICA DA VALVULA VS2212
  O:8.2: MOVE VALOR PARA SAIDA ANALOGICA DA VALVULA VS2213
  T4:27: ALARME PERDA DE COMUNICACAO COM EO2
  T4:25: ALARME PERDA DE COMUNICACAO COM EO1
  B9:5/1: MOVIMENTO DE RETORNO
  B20:5/8: PERFURATRIZ ATINGE FURO DE GUSA E ACIONA VS2217A (TRAVA PERFURATRIZ)
  B20:6/0: AVANCO ACIONA PORTA MARTELETE VS-2232
  B20:6/4: ACIONA VS-2233
  B20:5/12: RECUO ACIONA VS-2231
  B20:7/0: ROTATOR ACIONA VS-2236
  B20:6/8: MARTELO A FRENTE VS-2234
  B20:6/12: MANETE REVERSO VS-2235
  B20:7/4: SOPRO APENAS COM AR - ACIONA VS-2237
  B13:6/0: RESERV OLEO NIVEL BAIXO
  B13:7/0: RESERV OLEO TEMP ALTA
  B11:6/0: VALVUCCAO ABERTO
  B11:2/3: LOCAL
  B20:3/0: DESLIGA BOMBA
  B10:8/6: ALARMES VINDOS DAS ENTRADAS DIGITAIS
  B13:2/5: NIVEL DE OLEO MUITO BAIXO

REVISION NOTES
  17: CANHÃO 1 DIA 22/09/2013
  18: CANHÃO 1 EVERALDO

DATA TABLE (non-zero values as saved)
DATA B3
% B3:0 % 0X0000 0X0000 0X0000 0X0000 0X0000 0X0000 0X0001 0X0000 0X0000 0X0002
% B3:10 % 0X0000 0X0000 0X0000 0X0000 0X0000 0X0000 0X0000 0X0000 0X0000 0X0002
% B3:20 % 0X0000 0X0000 0X0000 0X0000 0X0000 0X0000 0X0000 0X0002 0X0000 0X0801
DATA T4
% .PRE .ACC %
% T4:0 % 6 0
% T4:1 % 4 0
% T4:2 % 5 0
% T4:3 % 10 0
% T4:4 % 40 0
% T4:5 % 25 19
% T4:6 % 20 0
% T4:7 % 5 0
% T4:8 % 1 0
% T4:9 % 40 0
% T4:10 % 10 0
% T4:11 % 10 0
% T4:12 % 10 0
% T4:13 % 10 0
% T4:14 % 20 0
% T4:15 % 10 0
% T4:16 % 10 0
% T4:17 % 1 0
% T4:18 % 5 0
% T4:19 % 5 0
% T4:20 % 5 0
% T4:21 % 5 0
% T4:22 % 60 60
% T4:23 % 50 50
% T4:24 % 50 0
% T4:25 % 30 0
% T4:26 % 50 0
% T4:27 % 30 30
% T4:28 % 30 30
% T4:29 % 3 0
% T4:31 % 2 0
% T4:32 % 2 0
% T4:33 % 5 0
% T4:34 % 5 0
% T4:35 % 20 20
% T4:36 % 1 0
% T4:37 % 1 0
% T4:38 % 2 0
% T4:39 % 1 0
% T4:40 % 20 20
% T4:41 % 5 0
% T4:42 % 2 0
% T4:43 % 60 0
% T4:44 % 60 0
% T4:45 % 5 1
% T4:50 % 1 0
% T4:51 % 3 0
% T4:60 % 500 500
% T4:195 % 5 0
% T4:198 % 20 0
% T4:200 % 10 0
DATA C5
% .PRE .ACC %
% C5:0 % 2 0
DATA R6
% .LEN .POS %
% R6:0 % 100 100
% R6:1 % 1 0
% R6:2 % 100 100
% R6:3 % 1 0
DATA N7
% N7:0 % 16 4 0
DATA F8
% F8:0 % 0 0 20 211.0111 1250.911
% F8:10 % 0 -50 -50 32.2375 0.984375
% F8:15 % 71.55 -625 -12.5 91.8875 100
% F8:20 % 0 0 45.33781 0 0
DATA B9
% B9:0 % 0X0002 0X0000 0X0000 0X0000 0X0000 0X0000 0X0000 0X0000 0X0000 0X0000
DATA B10
% B10:0 % 0X2082 0X0000 0X0000 0X0000 0X0000 0X0000 0X0000 0X0000 0X0000 0X0000
% B10:10 % 0X0000 0X1015 0X1000 0X4000 0X1400 0X0000
DATA B11
% B11:0 % 0X0000 0X0001 0X0001 0X0001 0X0001 0X0000 0X0002 0X8002 0X0000 0X0001
DATA B13
% B13:0 % 0X0006 0X0000 0X0000 0X0000 0X0000 0X0000 0X0000 0X0000 0X0000 0X0000
DATA N16
% N16:0 % 0 200 5 180 175 0 0 0 0 200
% N16:10 % 5 180 175 0 0 0 0 200 5 70
% N16:20 % 60 6 0 0 0 350 20 350 320 0
% N16:30 % 0 0 0 400 8 300 290 6 5 0
% N16:40 % 0 2500 100 240 230 52 42 0 0 400
% N16:50 % 8 350 320 0 0 0 0 100 1 100
% N16:60 % 97 70 65 0 150 350 0 350 350 0
% N16:70 % -100 0 0 0 0 0 0 0 0 0
DATA N17
% N17:0 % -50 -50 32 1 280 0 -13 92 100 -88
% N17:80 % 1 0 0 0 0 0 0 0 0 0
DATA B20
% B20:0 % 0X0000 0X0000 0X0000 0X0000 0X0000 0X0410 0X0000 0X0011 0X0000 0X0000
% B20:10 % 0X0100 0X0011
DATA B21
% B21:0 % 0X0000 0X1000 0X1100 0X0000 0X0000 0X0000 0X0000 0X1000 0X1100 0X0000
DATA N24
% N24:0 % 0 0 0 0 0 32 -24000 20000 -625 0
% N24:10 % 72 20 0 0 0 0 0 0 0 0
DATA N25
% N25:0 % 0 30800 0 0 0 0 0 0 0 0
DATA N26
% N26:0 % 0 0 6 11 133 0 0 0 5 0
% N26:10 % 0 12 0 0 12337 11824 12337 11824 12337 11824
% N26:20 % 49 0 0 0 0 0 0 0 0 0
DATA N27
% N27:0 % 0 0 8 13 133 0 0 0 5 0
% N27:10 % 0 16 0 0 12337 11824 12337 11824 12337 11824
% N27:20 % 49 0 0 0 0 0 0 0 0 0
DATA N29
% N29:0 % 0 350 350 0 -100 350 350 0 -100
DATA B31
% B31:0 % 0X0240 0X0200 0X0200 0X0000 0X0001 0X0000 0X0000 0X0000 0X0000 0X0000
% B31:10 % 0X0000 0X0000 0X0000 0X0000 0X0000 0X0000 0X0000 0X0000 0X0000 0X0002
% B31:20 % 0X0000 0X0000 0X0000 0X0001 0X0000 0X0002
DATA B33
% B33:0 % 0XC000 0X0000 0X0000 0X0000 0X0000 0X0000 0X0000 0X0000 0X0000 0X0000
% B33:20 % 0X0000 0X0000 0X0000 0X0000 0X0000 0X0001
DATA B39
% B39:0 % 0X0000 0X0000 0X0000 0X0000 0X0000 0X0002 0X0004 0X0004 0X0000 0X0000
DATA B41
% B41:0 % 0X0047 0X0052 0X0052 0X0000 0X0000 0X0000 0X0000 0X0000
